TYPE EL3204_DEV_CONFIG :
    STRUCT
   
        // Setpoint scaling
       	factor        : REAL := 0.01;  	
   
    END_STRUCT
END_TYPE

(* stored: Version 1.1.0.1, ProductVersion 3.1.4024.15
   DUT EL3204_DEV_CONFIG: Id {9239619a-8cb3-40c5-98b0-29cc10e27bcc} *)
